// Mitsubishi GX Works2 project: 230928-003-TIME ACION. 1 PULSO   PLC: Q03UDV

// task Task_01 (event TRUE, interval 0, priority 31): POU_01

PROGRAM POU_01
VAR
  RT0 : BOOL;  (* AASDF *)
END_VAR
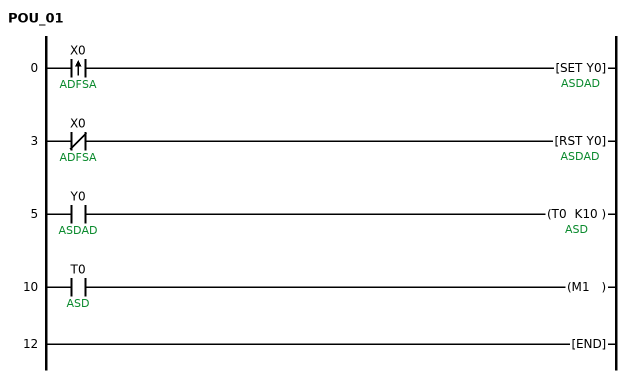
0     LDP     X0  ; ADFSA
      SET     Y0  ; ASDAD
3     LDI     X0  ; ADFSA
      RST     Y0  ; ASDAD
5     LD      Y0  ; ASDAD
      OUT     T0 K10  ; ASD
10    LD      T0  ; ASD
      OUT     M1
12    END
END_PROGRAM

// device comments not shown above
X1  ; ASDA
